// TIA Portal V18 export
DATA_BLOCK "MixingRatio_DB"   // DB137
VERSION : 0.1
// stored: AutoNumber true, DBAccessibleFromOPCUA true, InstanceOfName MixingRatio, InstanceOfType FB
"MixingRatio"
   // VAR_INPUT
   //    "Pump size A in ml" : Real;
   //    "Pump size B in ml" : Real;
   //    "Pump speed A_Max" : Real;
   //    "Pump speed B_Max" : Real;
   //    "Pump speed A_Passive" : Real;
   //    "Pump speed B_Passive" : Real;
   //    "Mixing ratio A100:B" : Real;
   //    "No.of Component" : Int;
   //    "Density A" : Real;
   //    "Density B" : Real;
   //    "Mixed Flowrate Set" : Real;
   //    "Flowrate Type" : Int;
   // END_VAR
   // VAR_OUTPUT
   //    "Maximum Flowrate A" : Real;
   //    "Maximum Flowrate B" : Real;
   //    "Maximum Flowrate A_Limited" : Real;
   //    "Maximum Flowrate B_Limited" : Real;
   //    "Maximum Flowrate Mixed" : Real;
   //    "Required flowrate A" : Real;
   //    "Required flowrate B" : Real;
   // END_VAR
   // VAR
   //    "Pump size A actual" : Real;
   //    "Pump size B actual" : Real;
   //    "Max flowrate A" : Real;
   //    "Max flowrate B" : Real;
   //    "Ratio margin B" : Real;
   //    "usable A flowrate per B ratio" : Real;
   //    "maximum mixed flowrate" : Real;
   //    "usable flowrate A per ratio" : Real;
   //    "usable flowrate B per ratio" : Real;
   //    "Flowrate difference A" : Real;
   //    "Flowrate difference B" : Real;
   //    "target flowrate A" : Real;
   //    "target flowrate B" : Real;
   // END_VAR
BEGIN
END_DATA_BLOCK
